PROGRAM prgHMILanguage
VAR
	tTrueLangIndex: UINT;
	tSizeOfLangRow: UINT;
	tSizeOfLangRowButtons: UINT;
	tStationNumberIndexLang: UINT;
	tScreenElementsPerPageLang: UINT;
	tNumElementsPerScreen: UINT;
	retval: UDINT;
END_VAR
VAR // added by the converter: edge detectors and wires of the graphical bodies
    _rt1, _rt2 : R_TRIG;
END_VAR

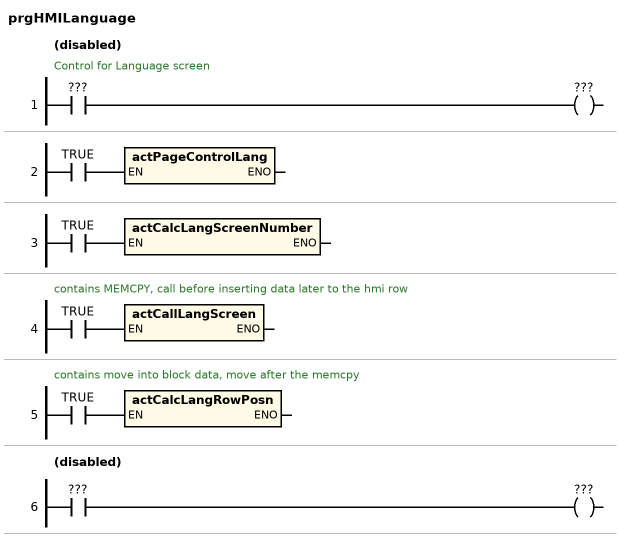
// NETWORK 1 (disabled)
// Control for Language screen
// ??? := ???;

// NETWORK 2
actPageControlLang();

// NETWORK 3
actCalcLangScreenNumber();

// NETWORK 4
// contains MEMCPY, call before inserting data later to the hmi row
actCallLangScreen();

// NETWORK 5
// contains move into block data, move after the memcpy
actCalcLangRowPosn();

// NETWORK 6 (disabled)
// ??? := ???;

ACTION actCalcLangRowPosn:
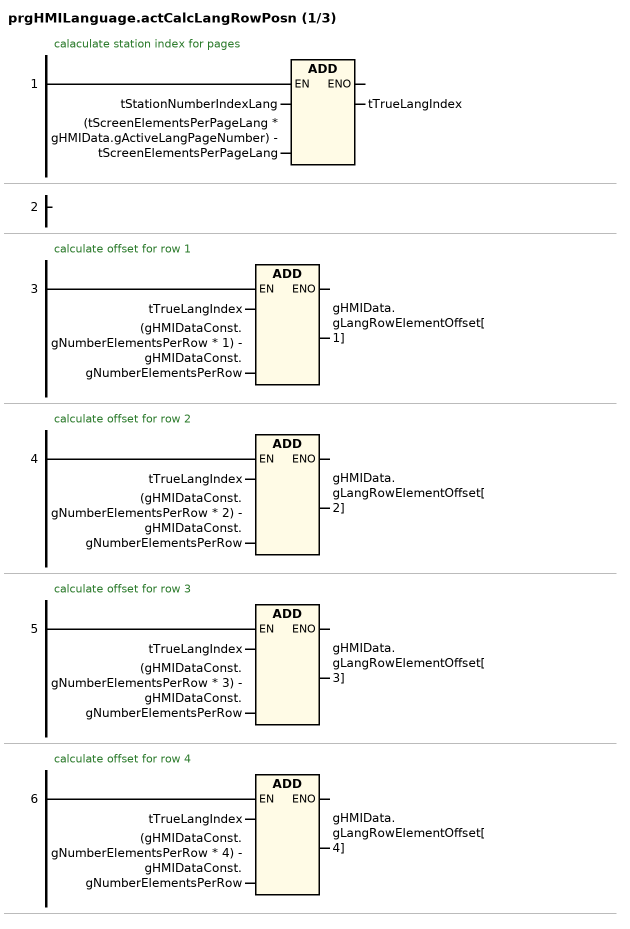
// NETWORK 1
// calaculate station index for pages
tTrueLangIndex := tStationNumberIndexLang + ((tScreenElementsPerPageLang * gHMIData.gActiveLangPageNumber) -  tScreenElementsPerPageLang);

// NETWORK 2

// NETWORK 3
// calculate offset for row 1
gHMIData.gLangRowElementOffset[1] := tTrueLangIndex + ((gHMIDataConst.gNumberElementsPerRow * 1) - gHMIDataConst.gNumberElementsPerRow);

// NETWORK 4
// calculate offset for row 2
gHMIData.gLangRowElementOffset[2] := tTrueLangIndex + ((gHMIDataConst.gNumberElementsPerRow * 2) - gHMIDataConst.gNumberElementsPerRow);

// NETWORK 5
// calculate offset for row 3
gHMIData.gLangRowElementOffset[3] := tTrueLangIndex + ((gHMIDataConst.gNumberElementsPerRow * 3) - gHMIDataConst.gNumberElementsPerRow);

// NETWORK 6
// calculate offset for row 4
gHMIData.gLangRowElementOffset[4] := tTrueLangIndex + ((gHMIDataConst.gNumberElementsPerRow * 4) - gHMIDataConst.gNumberElementsPerRow);

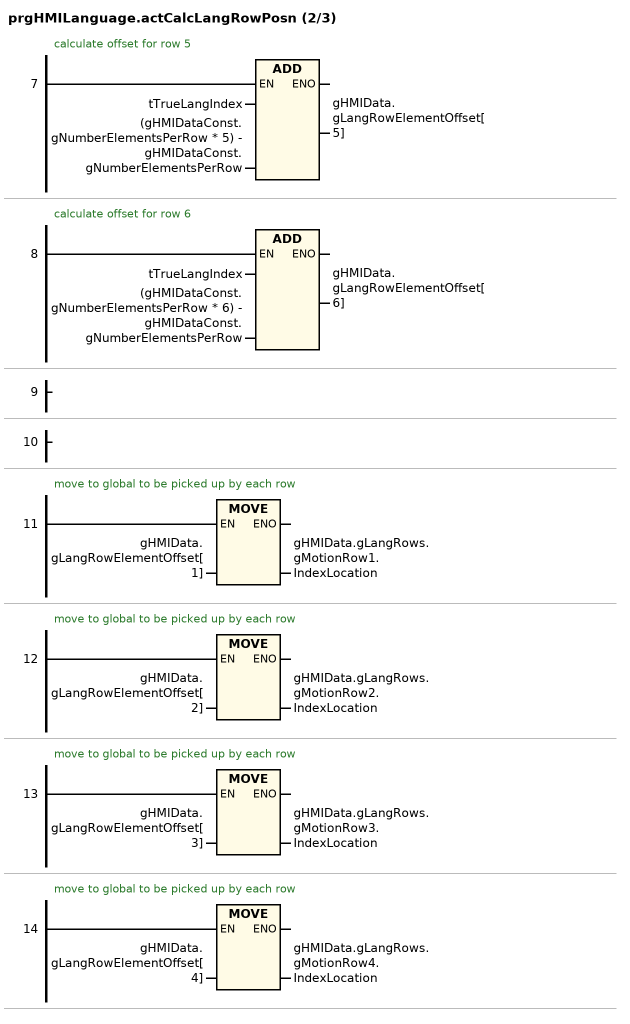
// NETWORK 7
// calculate offset for row 5
gHMIData.gLangRowElementOffset[5] := tTrueLangIndex + ((gHMIDataConst.gNumberElementsPerRow * 5) - gHMIDataConst.gNumberElementsPerRow);

// NETWORK 8
// calculate offset for row 6
gHMIData.gLangRowElementOffset[6] := tTrueLangIndex + ((gHMIDataConst.gNumberElementsPerRow * 6) - gHMIDataConst.gNumberElementsPerRow);

// NETWORK 9

// NETWORK 10

// NETWORK 11
// move to global to be picked up by each row
gHMIData.gLangRows.gMotionRow1.IndexLocation := gHMIData.gLangRowElementOffset[1];

// NETWORK 12
// move to global to be picked up by each row
gHMIData.gLangRows.gMotionRow2.IndexLocation := gHMIData.gLangRowElementOffset[2];

// NETWORK 13
// move to global to be picked up by each row
gHMIData.gLangRows.gMotionRow3.IndexLocation := gHMIData.gLangRowElementOffset[3];

// NETWORK 14
// move to global to be picked up by each row
gHMIData.gLangRows.gMotionRow4.IndexLocation := gHMIData.gLangRowElementOffset[4];

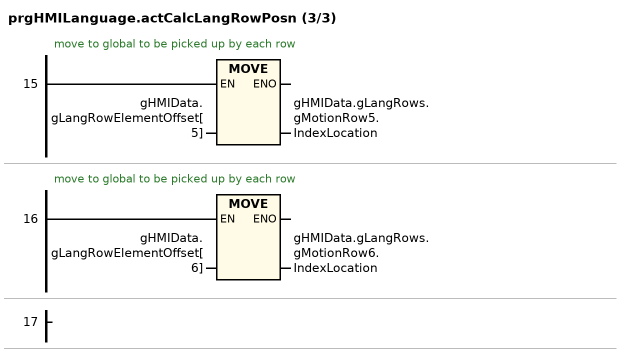
// NETWORK 15
// move to global to be picked up by each row
gHMIData.gLangRows.gMotionRow5.IndexLocation := gHMIData.gLangRowElementOffset[5];

// NETWORK 16
// move to global to be picked up by each row
gHMIData.gLangRows.gMotionRow6.IndexLocation := gHMIData.gLangRowElementOffset[6];

// NETWORK 17
END_ACTION

ACTION actCalcLangScreenNumber:
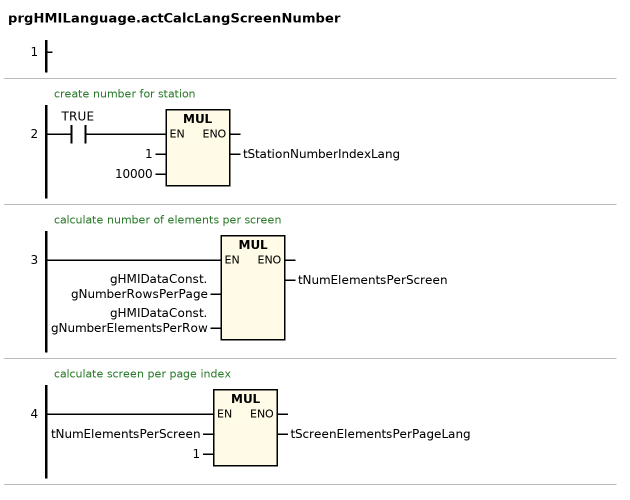
// NETWORK 1

// NETWORK 2
// create number for station
tStationNumberIndexLang := 1 * 10000;

// NETWORK 3
// calculate number of elements per screen
tNumElementsPerScreen := gHMIDataConst.gNumberRowsPerPage * gHMIDataConst.gNumberElementsPerRow;

// NETWORK 4
// calculate screen per page index
tScreenElementsPerPageLang := tNumElementsPerScreen * 1;
END_ACTION

ACTION actCallLangScreen:
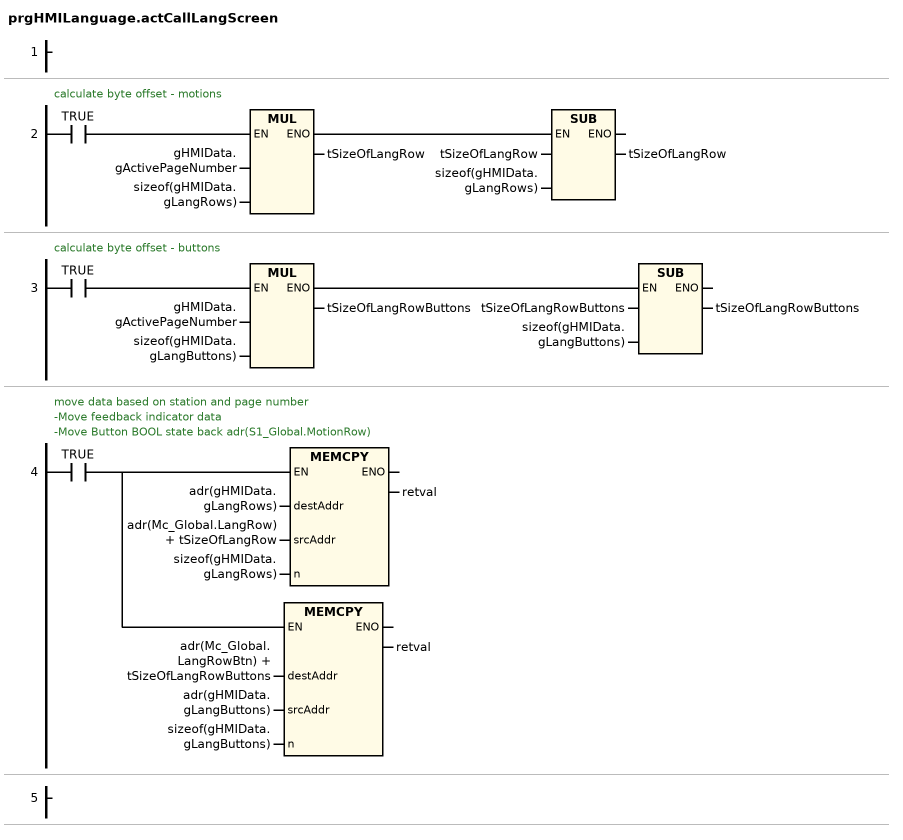
// NETWORK 1

// NETWORK 2
// calculate byte offset - motions
tSizeOfLangRow := gHMIData.gActivePageNumber * (sizeof(gHMIData.gLangRows));
tSizeOfLangRow := tSizeOfLangRow - (sizeof(gHMIData.gLangRows));

// NETWORK 3
// calculate byte offset - buttons
tSizeOfLangRowButtons := gHMIData.gActivePageNumber * (sizeof(gHMIData.gLangButtons));
tSizeOfLangRowButtons := tSizeOfLangRowButtons - (sizeof(gHMIData.gLangButtons));

// NETWORK 4
// move data based on station and page number
// -Move feedback indicator data
// -Move Button BOOL state back adr(S1_Global.MotionRow)
retval := MEMCPY(destAddr := adr(gHMIData.gLangRows), srcAddr := adr(Mc_Global.LangRow) + tSizeOfLangRow, n := sizeof(gHMIData.gLangRows));
retval := MEMCPY(destAddr := adr(Mc_Global.LangRowBtn) + tSizeOfLangRowButtons, srcAddr := adr(gHMIData.gLangButtons), n := sizeof(gHMIData.gLangButtons));

// NETWORK 5
END_ACTION

ACTION actPageControlLang:
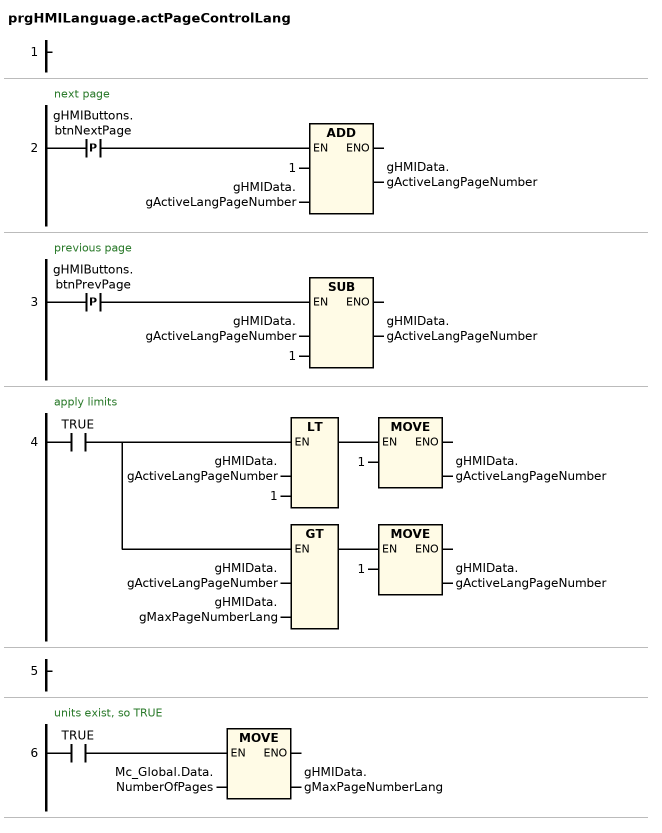
// NETWORK 1

// NETWORK 2
// next page
_rt1(CLK := gHMIButtons.btnNextPage);
IF _rt1.Q THEN gHMIData.gActiveLangPageNumber := 1 + gHMIData.gActiveLangPageNumber; END_IF

// NETWORK 3
// previous page
_rt2(CLK := gHMIButtons.btnPrevPage);
IF _rt2.Q THEN gHMIData.gActiveLangPageNumber := gHMIData.gActiveLangPageNumber - 1; END_IF

// NETWORK 4
// apply limits
IF gHMIData.gActiveLangPageNumber < 1 THEN gHMIData.gActiveLangPageNumber := 1; END_IF
IF gHMIData.gActiveLangPageNumber > gHMIData.gMaxPageNumberLang THEN gHMIData.gActiveLangPageNumber := 1; END_IF

// NETWORK 5

// NETWORK 6
// units exist, so TRUE
gHMIData.gMaxPageNumberLang := Mc_Global.Data.NumberOfPages;
END_ACTION

END_PROGRAM

(* stored: Version 1.1.0.1, ProductVersion 3.1.4024.12
   POU prgHMILanguage: Id {6b5cd21b-5048-4800-a15f-88aa66e2e3d4}, SpecialFunc None
   Action actCalcLangRowPosn: Id {ab5dd2f7-2246-4dc5-b157-18ed65fc115b}
   Action actCalcLangScreenNumber: Id {9bca8da3-1bd5-4f38-b00a-fdcf9a7a823e}
   Action actCallLangScreen: Id {efd40dd9-490d-4792-baef-abbd591fb521}
   Action actPageControlLang: Id {c30bf3f0-038c-458a-8f13-ea59d4c51a60} *)
